FUNCTION_BLOCK FB_Vereinzelung
VAR_INPUT
	// Steuervariablen
	bEnable : BOOL;
	bExecute : BOOL;
	
	// Hardware Eingänge
	bSensor1 : BOOL;	// Flasche in Kammer
	bSensor2 : BOOL;	// Flasche im Rohr
	bSensor3 : BOOL;	// Flaschenkopf
	bSensor4 : BOOL;	// Flasche am Fließband
END_VAR
VAR_OUTPUT
	// Steuervariable
	eState : eBetriebszustand;	

	//Hardware Ausgänge
	bGate1 : BOOL := FALSE;
	bGate2 : BOOL := FALSE;
END_VAR
VAR
	nState : INT := 100;
	fbTON : TON;
END_VAR

fbTON(IN:= , PT:= T#2S, Q=> , ET=> );
CASE nState OF
	100: // OFF
	eState := eBetriebszustand.OFF;
	
	IF bSensor1 AND bEnable THEN
		nState := 21; //READY
	ELSIF bEnable THEN
		nState := 0; // INIT 
	END_IF
	
	0: // INIT-Kammer leer
	eState := eBetriebszustand.INIT;
	
	bGate1 := FALSE;
	bGate2 := FALSE;
	
	IF bSensor2 THEN
		nState := 1; // Oben öffnen
	END_IF
	
	1: // INIT-Oben öffnen
	eState := eBetriebszustand.INIT;
	
	bGate1 := TRUE;
	bGate2 := FALSE;
	
	IF bSensor1 = TRUE THEN
		nState := 2; // Oben schließen
	END_IF
	
	2: // INIT-Oben schließen
	eState := eBetriebszustand.INIT;
	
	bGate1 := FALSE;
	bGate2 := FALSE;
	fbTON.IN := TRUE;
	
	IF fbTON.Q AND bSensor1 THEN
		fbTON.IN := FALSE;
		nState := 21; // READY
	END_IF
	
	21: // READY
	eState := eBetriebszustand.READY;
	bGate1 := FALSE;
	bGate2 := FALSE;
	
	IF bExecute THEN
		nState := 3; // Unten öffnen
	END_IF
	
	3: // PROD-Unten öffnen
	eState := eBetriebszustand.PROD;
	
	bGate1 := FALSE;
	bGate2 := TRUE;
	
	IF bSensor4 THEN
		nState := 4; //Unten schließen
	END_IF
	
	4: // PROD-Unten schließen
	eState := eBetriebszustand.PROD;
	
	bGate1 := FALSE;
	bGate2 := FALSE;
	fbTON.IN := TRUE;
	
	IF fbTON.Q THEN
		fbTON.IN := FALSE;
		nState := 41; // DONE
	END_IF
	
	41: // DONE
	eState := eBetriebszustand.DONE;
	
	bGate1 := FALSE;
	bGate2 := FALSE;
	
	IF NOT bExecute THEN
		nState := 0; // Kammer leer
	END_IF
	
END_CASE

END_FUNCTION_BLOCK

(* stored: Version 1.1.0.1, ProductVersion 3.1.4024.15
   POU FB_Vereinzelung: Id {0b53d581-c894-4398-8b7b-4ddadede748e}, SpecialFunc None *)
